// TIA Portal V15.1 export
// export: Created 2024-06-21T08:41:10.2216072Z, ExportSetting WithDefaults, DisplayName Totally Integrated Automation Portal, DisplayVersion V15.1 Update 5, DisplayName TIA Portal Openness, DisplayVersion V15.1 Update 5, DisplayName SINAMICS Startdrive Advanced, DisplayVersion V15.1, DisplayName G130, G150, S120, S150, SINAMICS MV, S210, DisplayVersion V15.1, DisplayName G110M, G120, G120C, G120D, G120P, DisplayVersion V15.1, DisplayName STEP 7 Professional, DisplayVersion V15.1 Update 5, DisplayName STEP 7 Safety, DisplayVersion V15.1, DisplayName WinCC Professional, DisplayVersion V15.1 Update 5, DisplayName SIMATIC Visualization Architect, DisplayVersion V15.1
FUNCTION "LGBRoller2W2S-C-Config" : Void   // FC6608, FBD
TITLE = LRoller2W2S-C-Config / LGBRoller2W2S-C-Config
{ S7_Optimized_Access := 'TRUE' }
AUTHOR : VCC
FAMILY : Config
NAME : Bit2Word
VERSION : 0.1
// =============================================================================
// Moves the 16 input bits to one output integer 
// =============================================================================
// stored: AutoNumber false, IsIECCheckEnabled false, SetENOAutomatically False, UDAEnableTagReadback false
   VAR_INPUT
      C_DeadEnd : Bool;   // Dead End Disable Positiong Fault / Config
      C_StopDetSetUsed : Bool;   // Config
      C_LowSpeedDetSetUsed : Bool;   // Config
      C_LowSpeedDetSetConstOn : Bool;   // Config
      C_LowSpeedDetResUsed : Bool;   // Config
      C_LowSpeedDetResConstOn : Bool;   // Config
      C_StopDetResUsed : Bool;   // Config
      C_OccupiedDetUsed : Bool;   // Config
      C_TrainActivatedSet : Bool;   // Config
      C_TrfInSetUsed : Bool;   // Config
      C_TrfInSetInLowSpeed : Bool;   // Input 4 / Transfer In Set ALL the time in low speed / Transfer In Set Used
      C_TrfOutSetUsed : Bool;   // Config
      C_TrfOutSetInLowSpeed : Bool;   // Input 5 / Transfer Out Set ALL the time in low speed / Transfer Out Reset Used
      C_TrainActivatedRes : Bool;   // Config
      C_TrfInResUsed : Bool;   // Config
      C_TrfInResInLowSpeed : Bool;   // Input 13 / Transfer In Reset ALL the time in low speed / Transfer In Reset Used
      C_TrfOutResUsed : Bool;   // Config
      C_TrfOutResInLowSpeed : Bool;   // Input 14 / Transfer Out Reset ALL the time in low speed / Transfer Out Reset Used
      C_TrspNoLowSpeed : Bool;   // Config / Transfer don't go to low speed because the next roller is ready to receive
      C_SafetySwNc : Bool;   // Config
      C_SafetySwUsed : Bool;   // Config
      C_MotorProtectionNc : Bool;   // Config
      C_MotorProtectionUsed : Bool;   // Config
      C_BrakeProtectionNc : Bool;   // Config
      C_BrakeProtectionUsed : Bool;   // Config
      C_ReleaseBrakeUsed : Bool;   // Config
      C_MotionStopUsed : Bool;   // Config
      C_EnableAlarmHW : Bool;   // Enable Alarm hardware (e.g. safetyswitch, motorprotector, detections) / Config
      C_EnableAlarmTransfer : Bool;   // Enable Alarm transfer (e.g. Transfer in , transfer out) / Config
      C_TrfMaxTime : DInt;   // Max allowed transfertime (millisec) / Config
      C_TrfMaxTimeAfterOvertime : DInt;   // Max allowed transfertime after overtime (millisec)
   END_VAR
   VAR_IN_OUT
      IO_Config : "RollerConvConfig";   // Config
   END_VAR
BEGIN

REGION Network 1: **** 1 - Inputs **** Move Config
   // Move Config
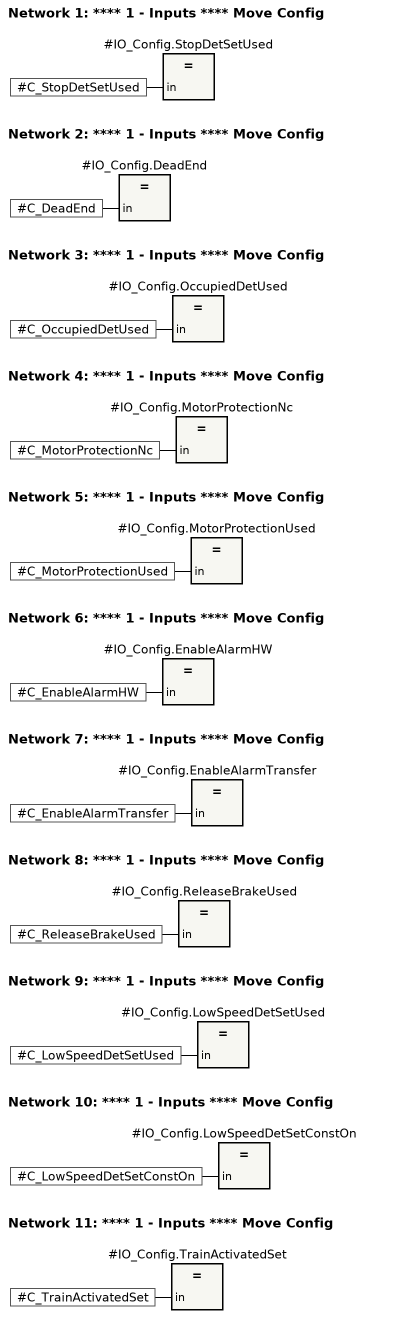
   #IO_Config.StopDetSetUsed := #C_StopDetSetUsed;
END_REGION

REGION Network 2: **** 1 - Inputs **** Move Config
   // Move Config
   #IO_Config.DeadEnd := #C_DeadEnd;
END_REGION

REGION Network 3: **** 1 - Inputs **** Move Config
   // Move Config
   #IO_Config.OccupiedDetUsed := #C_OccupiedDetUsed;
END_REGION

REGION Network 4: **** 1 - Inputs **** Move Config
   // Move Config
   #IO_Config.MotorProtectionNc := #C_MotorProtectionNc;
END_REGION

REGION Network 5: **** 1 - Inputs **** Move Config
   // Move Config
   #IO_Config.MotorProtectionUsed := #C_MotorProtectionUsed;
END_REGION

REGION Network 6: **** 1 - Inputs **** Move Config
   // Move Config
   #IO_Config.EnableAlarmHW := #C_EnableAlarmHW;
END_REGION

REGION Network 7: **** 1 - Inputs **** Move Config
   // Move Config
   #IO_Config.EnableAlarmTransfer := #C_EnableAlarmTransfer;
END_REGION

REGION Network 8: **** 1 - Inputs **** Move Config
   // Move Config
   #IO_Config.ReleaseBrakeUsed := #C_ReleaseBrakeUsed;
END_REGION

REGION Network 9: **** 1 - Inputs **** Move Config
   // Move Config
   #IO_Config.LowSpeedDetSetUsed := #C_LowSpeedDetSetUsed;
END_REGION

REGION Network 10: **** 1 - Inputs **** Move Config
   // Move Config
   #IO_Config.LowSpeedDetSetConstOn := #C_LowSpeedDetSetConstOn;
END_REGION

REGION Network 11: **** 1 - Inputs **** Move Config
   // Move Config
   #IO_Config.TrainActivatedSet := #C_TrainActivatedSet;
END_REGION

REGION Network 12: **** 1 - Inputs **** Move Config
   // Move Config
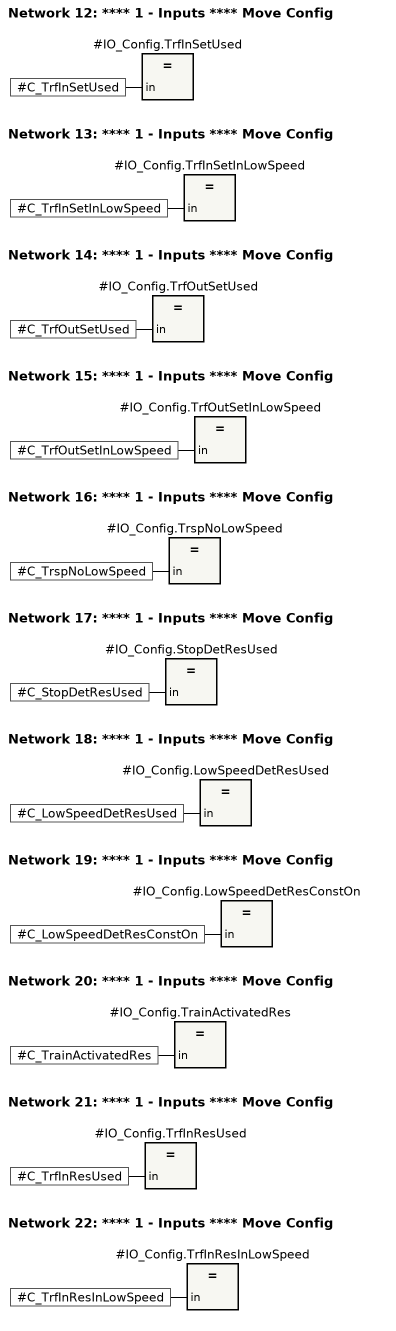
   #IO_Config.TrfInSetUsed := #C_TrfInSetUsed;
END_REGION

REGION Network 13: **** 1 - Inputs **** Move Config
   // Move Config
   #IO_Config.TrfInSetInLowSpeed := #C_TrfInSetInLowSpeed;
END_REGION

REGION Network 14: **** 1 - Inputs **** Move Config
   // Move Config
   #IO_Config.TrfOutSetUsed := #C_TrfOutSetUsed;
END_REGION

REGION Network 15: **** 1 - Inputs **** Move Config
   // Move Config
   #IO_Config.TrfOutSetInLowSpeed := #C_TrfOutSetInLowSpeed;
END_REGION

REGION Network 16: **** 1 - Inputs **** Move Config
   // Move Config
   #IO_Config.TrspNoLowSpeed := #C_TrspNoLowSpeed;
END_REGION

REGION Network 17: **** 1 - Inputs **** Move Config
   // Move Config
   #IO_Config.StopDetResUsed := #C_StopDetResUsed;
END_REGION

REGION Network 18: **** 1 - Inputs **** Move Config
   // Move Config
   #IO_Config.LowSpeedDetResUsed := #C_LowSpeedDetResUsed;
END_REGION

REGION Network 19: **** 1 - Inputs **** Move Config
   // Move Config
   #IO_Config.LowSpeedDetResConstOn := #C_LowSpeedDetResConstOn;
END_REGION

REGION Network 20: **** 1 - Inputs **** Move Config
   // Move Config
   #IO_Config.TrainActivatedRes := #C_TrainActivatedRes;
END_REGION

REGION Network 21: **** 1 - Inputs **** Move Config
   // Move Config
   #IO_Config.TrfInResUsed := #C_TrfInResUsed;
END_REGION

REGION Network 22: **** 1 - Inputs **** Move Config
   // Move Config
   #IO_Config.TrfInResInLowSpeed := #C_TrfInResInLowSpeed;
END_REGION

REGION Network 23: **** 1 - Inputs **** Move Config
   // Move Config
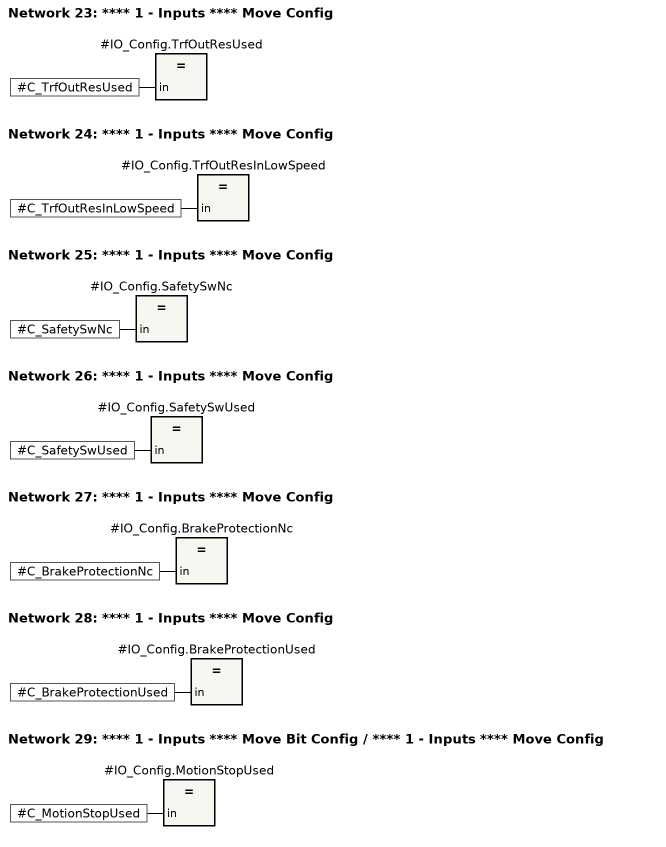
   #IO_Config.TrfOutResUsed := #C_TrfOutResUsed;
END_REGION

REGION Network 24: **** 1 - Inputs **** Move Config
   // Move Config
   #IO_Config.TrfOutResInLowSpeed := #C_TrfOutResInLowSpeed;
END_REGION

REGION Network 25: **** 1 - Inputs **** Move Config
   // Move Config
   #IO_Config.SafetySwNc := #C_SafetySwNc;
END_REGION

REGION Network 26: **** 1 - Inputs **** Move Config
   // Move Config
   #IO_Config.SafetySwUsed := #C_SafetySwUsed;
END_REGION

REGION Network 27: **** 1 - Inputs **** Move Config
   // Move Config
   #IO_Config.BrakeProtectionNc := #C_BrakeProtectionNc;
END_REGION

REGION Network 28: **** 1 - Inputs **** Move Config
   // Move Config
   #IO_Config.BrakeProtectionUsed := #C_BrakeProtectionUsed;
END_REGION

REGION Network 29: **** 1 - Inputs **** Move Bit Config / **** 1 - Inputs **** Move Config
   // Move Bit Config / Move Config
   #IO_Config.MotionStopUsed := #C_MotionStopUsed;
END_REGION

NETWORK
TITLE = **** 8 - Outputs **** Move Config UDT / **** 1 - Inputs **** Move Config UDT
// Move Config
      L     #C_TrfMaxTime;
      T     #IO_Config.TrfMaxTime;
      L     #C_TrfMaxTimeAfterOvertime;
      T     #IO_Config.TrfMaxTimeAfterOvertime;

END_FUNCTION
